DATA_BLOCK "EM_Rotator_Brake_DB"
{ S7_Optimized_Access := 'TRUE' }
VERSION : 0.1
"EM_Rotator_Brake"
BEGIN
END_DATA_BLOCK
